PROGRAM XDrive_Manager
VAR
	XDrive_Offset: LREAL; //general offset of the encoder value
	ExtraSensorInput: TAxSensorModule; // compressed FUN for exteriour sensor inputs. temp, edge, jog stops
	SpecialOperations: TAxSpecialOperationModule; //compressed FUN for the special operation commands. 
	AxisCoupleIN: TAxCoupleModule; //connects to the AX_Couple_out of the manager from the next axis. NOT MASTER/SLAVE
	ErrorWordArray: WORD; //build a array of words that act as a cluster of error watching variables. each step in array will be one axis. differant values of the word for each axis mean a differant error. 
	JogStop: LREAL := 1E100 ; // a stopping point using the jog system to signify it is in the right spot. Need to have the LimitPosJOG adjusted after to compensate for the next space.
	DriveCMD_1: DriveCMDShortCUT; //extra system for the FB to make it easy to read.
	ASPshortCut_1: ASPshortCUT;  // same as above
	FB_XDrivePotIN: FB_AnalogIn;
	ACHSRETURN_Xdrive: TAxReturn;
	FB_XDriveRipCutSpeed: FB_AnalogIn;
END_VAR

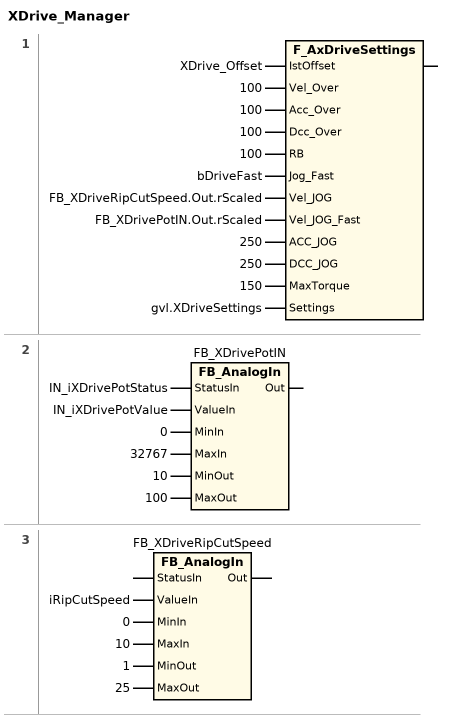
// NETWORK 1
F_AxDriveSettings(IstOffset := XDrive_Offset, Vel_Over := 100, Acc_Over := 100, Dcc_Over := 100, RB := 100, Jog_Fast := bDriveFast, Vel_JOG := FB_XDriveRipCutSpeed.Out.rScaled, Vel_JOG_Fast := FB_XDrivePotIN.Out.rScaled, ACC_JOG := 250, DCC_JOG := 250, MaxTorque := 150, Settings := gvl.XDriveSettings);

// NETWORK 2
FB_XDrivePotIN(
    StatusIn := IN_iXDrivePotStatus,
    ValueIn := IN_iXDrivePotValue,
    MinIn := 0,
    MaxIn := 32767,
    MinOut := 10,
    MaxOut := 100); // FB_AnalogIn

// NETWORK 3
FB_XDriveRipCutSpeed(ValueIn := iRipCutSpeed, MinIn := 0, MaxIn := 10, MinOut := 1, MaxOut := 25); // FB_AnalogIn

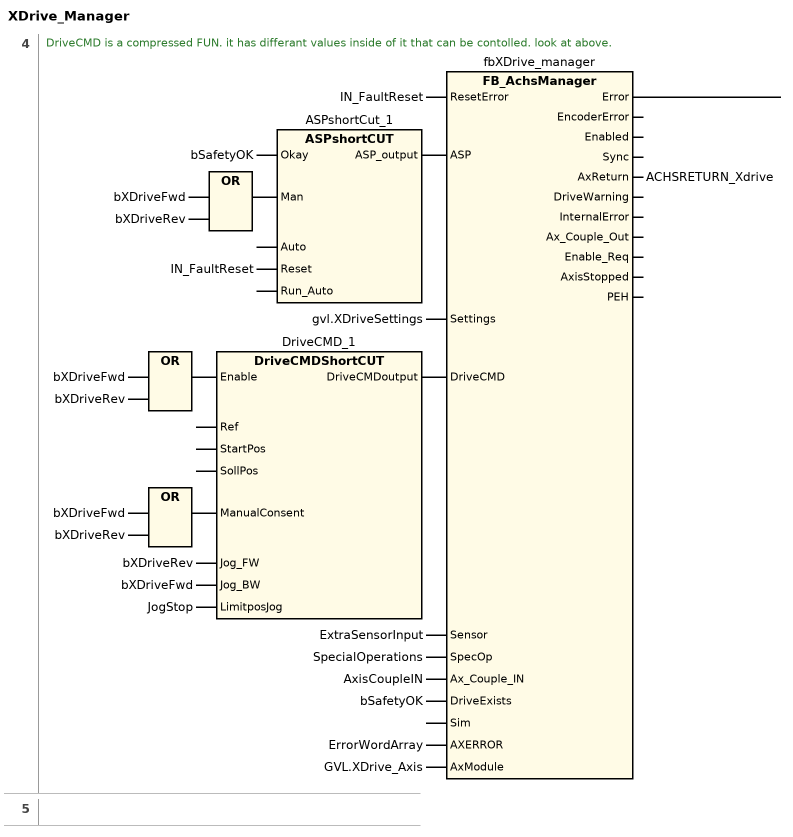
// NETWORK 4
// DriveCMD is a compressed FUN. it has differant values inside of it that can be contolled. look at above.
ASPshortCut_1(Okay := bSafetyOK, Man := bXDriveFwd OR bXDriveRev, Reset := IN_FaultReset); // ASPshortCUT
DriveCMD_1(
    Enable := bXDriveFwd OR bXDriveRev,
    ManualConsent := bXDriveFwd OR bXDriveRev,
    Jog_FW := bXDriveRev,
    Jog_BW := bXDriveFwd,
    LimitposJog := JogStop); // DriveCMDShortCUT
fbXDrive_manager(
    ResetError := IN_FaultReset,
    ASP := ASPshortCut_1.ASP_output,
    Settings := gvl.XDriveSettings,
    DriveCMD := DriveCMD_1.DriveCMDoutput,
    Sensor := ExtraSensorInput,
    SpecOp := SpecialOperations,
    Ax_Couple_IN := AxisCoupleIN,
    DriveExists := bSafetyOK,
    AXERROR := ErrorWordArray,
    AxModule := GVL.XDrive_Axis,
    AxReturn => ACHSRETURN_Xdrive); // FB_AchsManager

// NETWORK 5

END_PROGRAM

(* stored: Version 1.1.0.1, ProductVersion 3.1.4024.15
   POU XDrive_Manager: Id {c1103842-8e3f-4779-b875-a767321bf7ff}, SpecialFunc None *)
